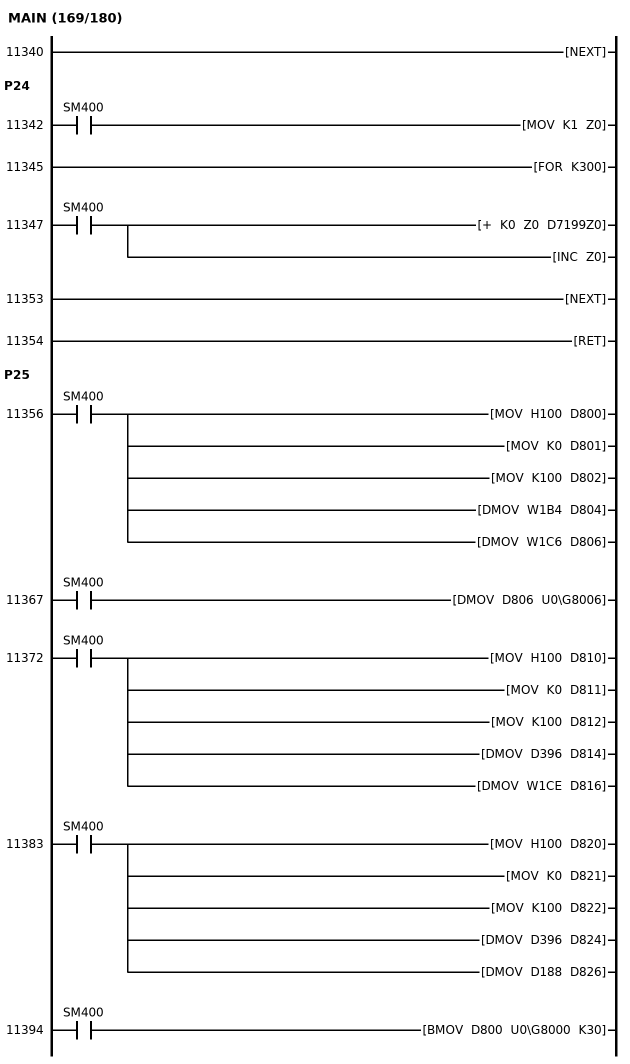
[picture p168: ladder of MAIN, rungs at steps 11340 to 11394]
11340 NEXT
      P24
11342 LD      SM400
      MOV     K1 Z0
11345 FOR     K300
11347 LD      SM400
      +       K0 Z0 D7199Z0
      INC     Z0
11353 NEXT
11354 RET
      P25
11356 LD      SM400
      MOV     H100 D800
      MOV     K0 D801
      MOV     K100 D802
      DMOV    W1B4 D804
      DMOV    W1C6 D806
11367 LD      SM400
      DMOV    D806 U0\G8006
11372 LD      SM400
      MOV     H100 D810
      MOV     K0 D811
      MOV     K100 D812
      DMOV    D396 D814
      DMOV    W1CE D816
11383 LD      SM400
      MOV     H100 D820
      MOV     K0 D821
      MOV     K100 D822
      DMOV    D396 D824
      DMOV    D188 D826
11394 LD      SM400
      BMOV    D800 U0\G8000 K30
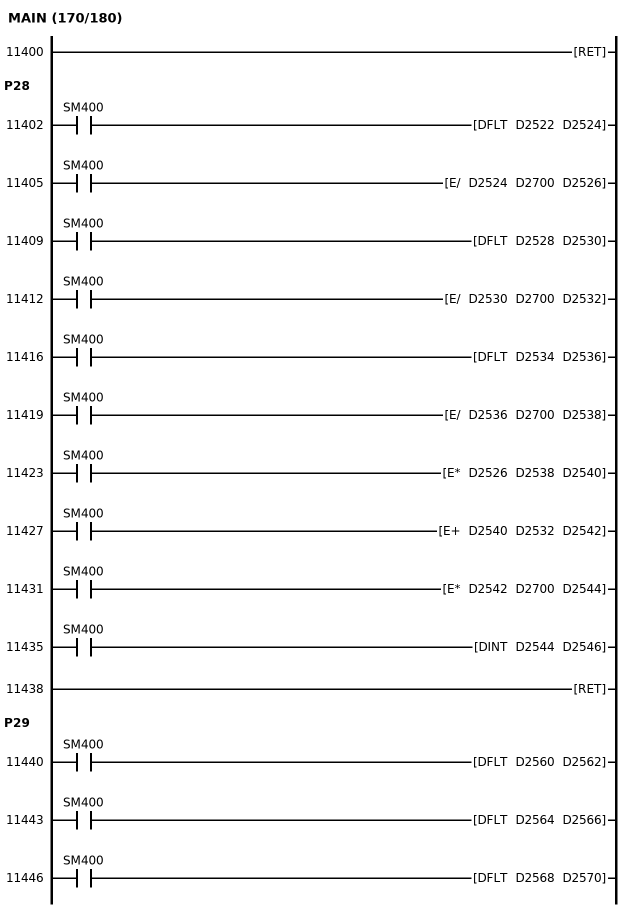
11400 RET
      P28
11402 LD      SM400
      DFLT    D2522 D2524
11405 LD      SM400
      E/      D2524 D2700 D2526
11409 LD      SM400
      DFLT    D2528 D2530
11412 LD      SM400
      E/      D2530 D2700 D2532
11416 LD      SM400
      DFLT    D2534 D2536
11419 LD      SM400
      E/      D2536 D2700 D2538
11423 LD      SM400
      E*      D2526 D2538 D2540
11427 LD      SM400
      E+      D2540 D2532 D2542
11431 LD      SM400
      E*      D2542 D2700 D2544
11435 LD      SM400
      DINT    D2544 D2546
11438 RET
      P29
11440 LD      SM400
      DFLT    D2560 D2562
11443 LD      SM400
      DFLT    D2564 D2566
11446 LD      SM400
      DFLT    D2568 D2570
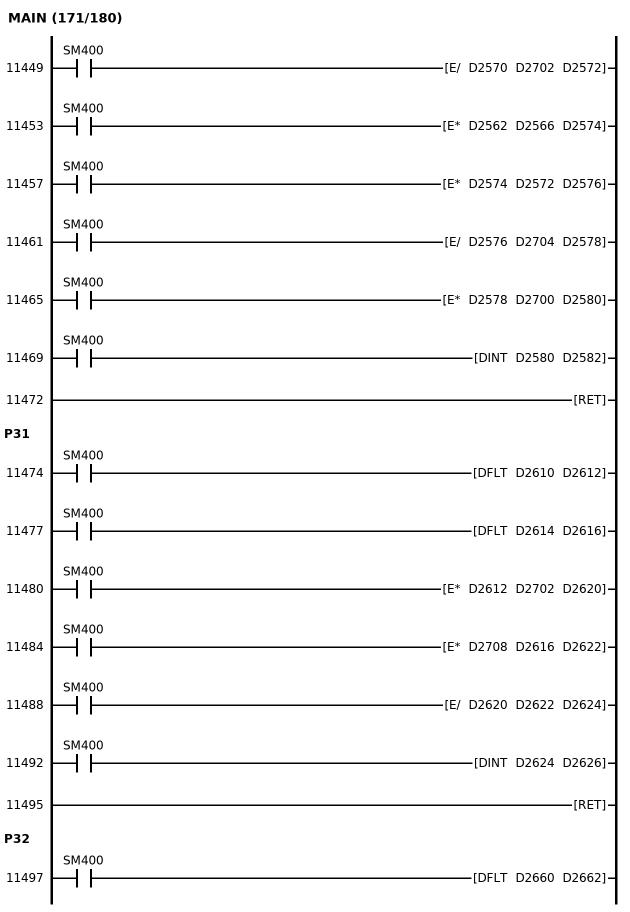
11449 LD      SM400
      E/      D2570 D2702 D2572
11453 LD      SM400
      E*      D2562 D2566 D2574
11457 LD      SM400
      E*      D2574 D2572 D2576
11461 LD      SM400
      E/      D2576 D2704 D2578
11465 LD      SM400
      E*      D2578 D2700 D2580
11469 LD      SM400
      DINT    D2580 D2582
11472 RET
      P31
11474 LD      SM400
      DFLT    D2610 D2612
11477 LD      SM400
      DFLT    D2614 D2616
11480 LD      SM400
      E*      D2612 D2702 D2620
11484 LD      SM400
      E*      D2708 D2616 D2622
11488 LD      SM400
      E/      D2620 D2622 D2624
11492 LD      SM400
      DINT    D2624 D2626
11495 RET
      P32
11497 LD      SM400
      DFLT    D2660 D2662
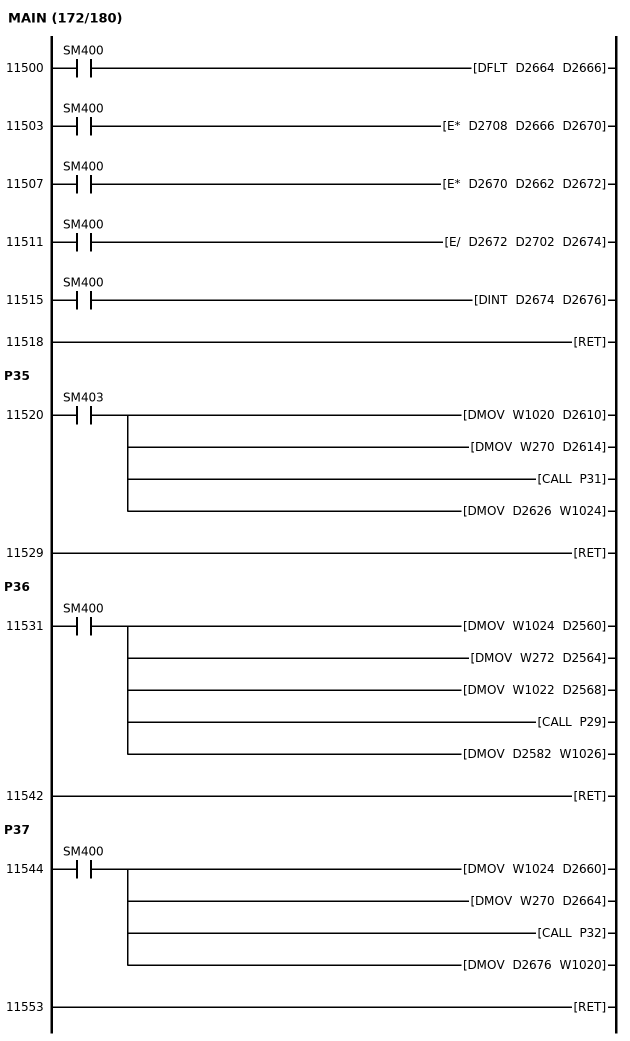
11500 LD      SM400
      DFLT    D2664 D2666
11503 LD      SM400
      E*      D2708 D2666 D2670
11507 LD      SM400
      E*      D2670 D2662 D2672
11511 LD      SM400
      E/      D2672 D2702 D2674
11515 LD      SM400
      DINT    D2674 D2676
11518 RET
      P35
11520 LD      SM403
      DMOV    W1020 D2610
      DMOV    W270 D2614
      CALL    P31
      DMOV    D2626 W1024
11529 RET
      P36
11531 LD      SM400
      DMOV    W1024 D2560
      DMOV    W272 D2564
      DMOV    W1022 D2568
      CALL    P29
      DMOV    D2582 W1026
11542 RET
      P37
11544 LD      SM400
      DMOV    W1024 D2660
      DMOV    W270 D2664
      CALL    P32
      DMOV    D2676 W1020
11553 RET
      P40
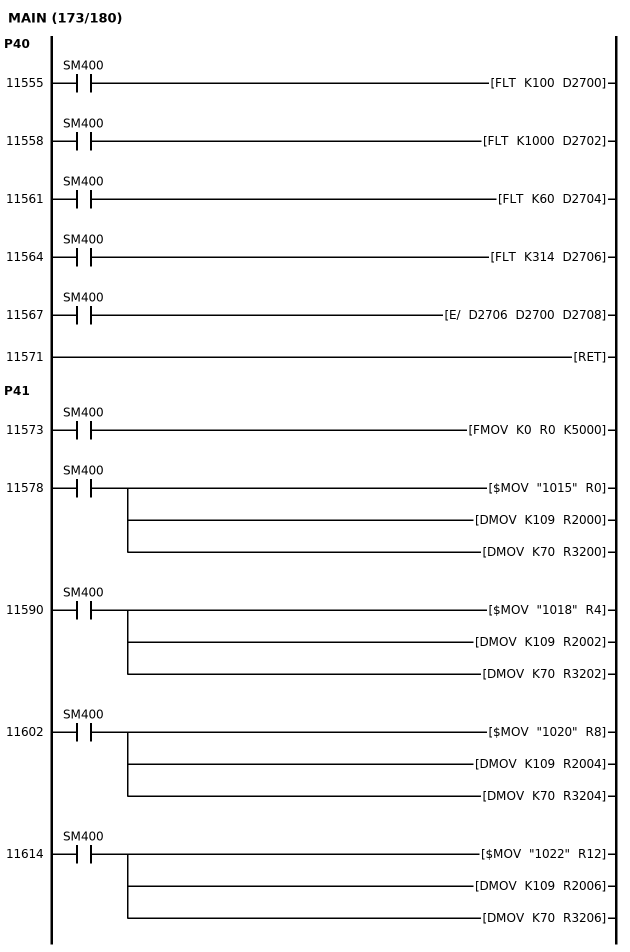
11555 LD      SM400
      FLT     K100 D2700
11558 LD      SM400
      FLT     K1000 D2702
11561 LD      SM400
      FLT     K60 D2704
11564 LD      SM400
      FLT     K314 D2706
11567 LD      SM400
      E/      D2706 D2700 D2708
11571 RET
      P41
11573 LD      SM400
      FMOV    K0 R0 K5000
11578 LD      SM400
      $MOV    "1015" R0
      DMOV    K109 R2000
      DMOV    K70 R3200
11590 LD      SM400
      $MOV    "1018" R4
      DMOV    K109 R2002
      DMOV    K70 R3202
11602 LD      SM400
      $MOV    "1020" R8
      DMOV    K109 R2004
      DMOV    K70 R3204
11614 LD      SM400
      $MOV    "1022" R12
      DMOV    K109 R2006
      DMOV    K70 R3206
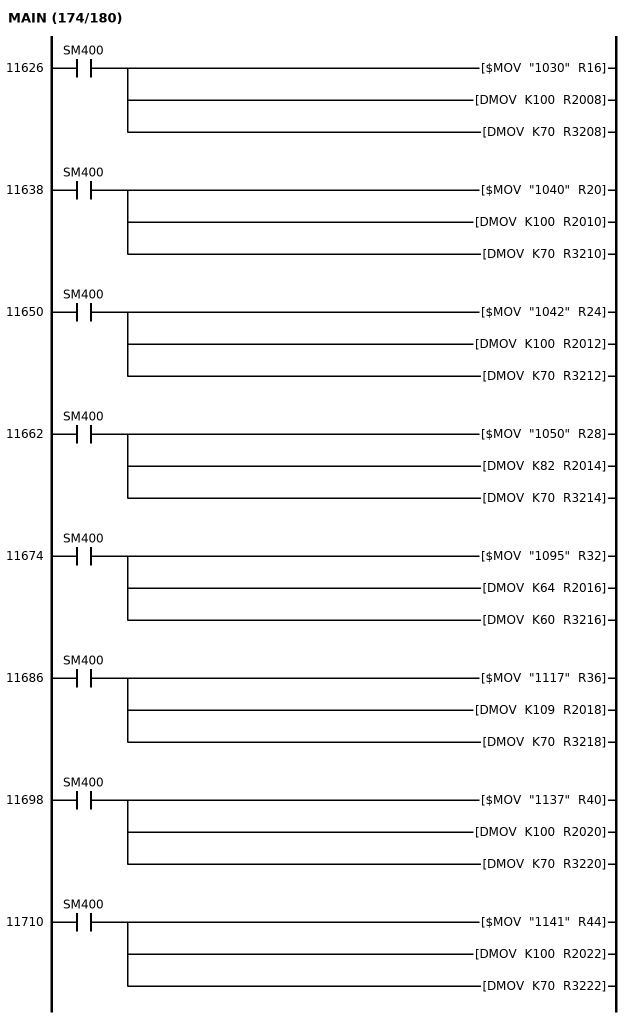
11626 LD      SM400
      $MOV    "1030" R16
      DMOV    K100 R2008
      DMOV    K70 R3208
11638 LD      SM400
      $MOV    "1040" R20
      DMOV    K100 R2010
      DMOV    K70 R3210
11650 LD      SM400
      $MOV    "1042" R24
      DMOV    K100 R2012
      DMOV    K70 R3212
11662 LD      SM400
      $MOV    "1050" R28
      DMOV    K82 R2014
      DMOV    K70 R3214
11674 LD      SM400
      $MOV    "1095" R32
      DMOV    K64 R2016
      DMOV    K60 R3216
11686 LD      SM400
      $MOV    "1117" R36
      DMOV    K109 R2018
      DMOV    K70 R3218
11698 LD      SM400
      $MOV    "1137" R40
      DMOV    K100 R2020
      DMOV    K70 R3220
11710 LD      SM400
      $MOV    "1141" R44
      DMOV    K100 R2022
      DMOV    K70 R3222
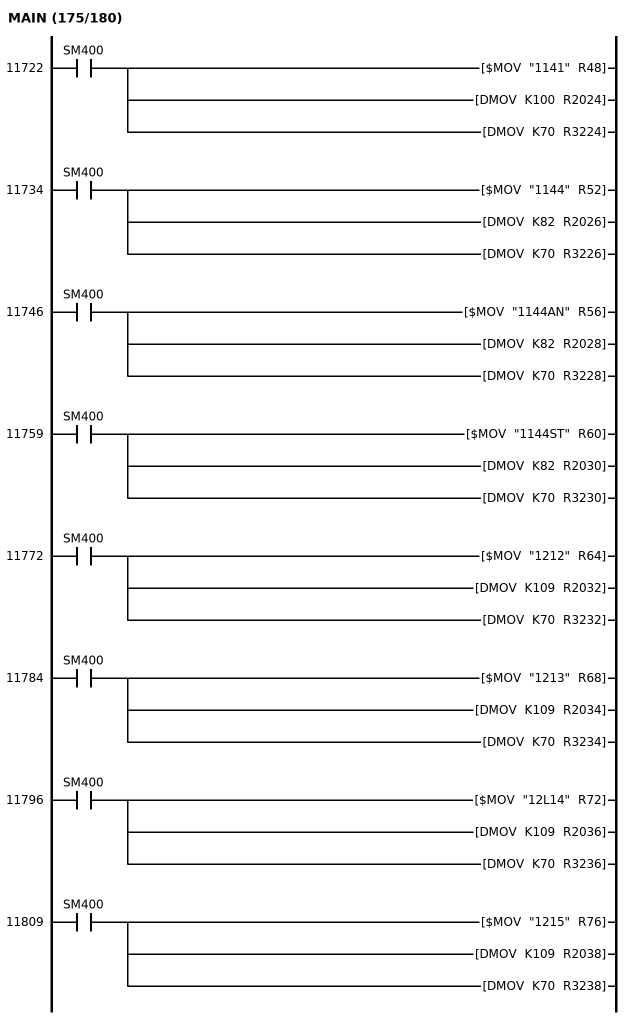
11722 LD      SM400
      $MOV    "1141" R48
      DMOV    K100 R2024
      DMOV    K70 R3224
11734 LD      SM400
      $MOV    "1144" R52
      DMOV    K82 R2026
      DMOV    K70 R3226
11746 LD      SM400
      $MOV    "1144AN" R56
      DMOV    K82 R2028
      DMOV    K70 R3228
11759 LD      SM400
      $MOV    "1144ST" R60
      DMOV    K82 R2030
      DMOV    K70 R3230
11772 LD      SM400
      $MOV    "1212" R64
      DMOV    K109 R2032
      DMOV    K70 R3232
11784 LD      SM400
      $MOV    "1213" R68
      DMOV    K109 R2034
      DMOV    K70 R3234
11796 LD      SM400
      $MOV    "12L14" R72
      DMOV    K109 R2036
      DMOV    K70 R3236
11809 LD      SM400
      $MOV    "1215" R76
      DMOV    K109 R2038
      DMOV    K70 R3238
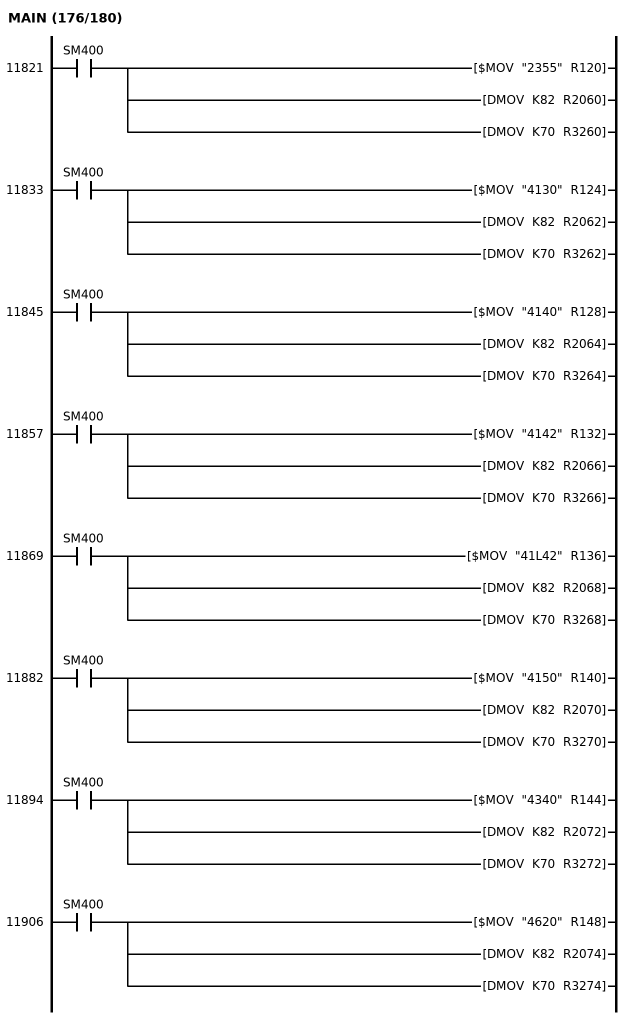
11821 LD      SM400
      $MOV    "2355" R120
      DMOV    K82 R2060
      DMOV    K70 R3260
11833 LD      SM400
      $MOV    "4130" R124
      DMOV    K82 R2062
      DMOV    K70 R3262
11845 LD      SM400
      $MOV    "4140" R128
      DMOV    K82 R2064
      DMOV    K70 R3264
11857 LD      SM400
      $MOV    "4142" R132
      DMOV    K82 R2066
      DMOV    K70 R3266
11869 LD      SM400
      $MOV    "41L42" R136
      DMOV    K82 R2068
      DMOV    K70 R3268
11882 LD      SM400
      $MOV    "4150" R140
      DMOV    K82 R2070
      DMOV    K70 R3270
11894 LD      SM400
      $MOV    "4340" R144
      DMOV    K82 R2072
      DMOV    K70 R3272
11906 LD      SM400
      $MOV    "4620" R148
      DMOV    K82 R2074
      DMOV    K70 R3274
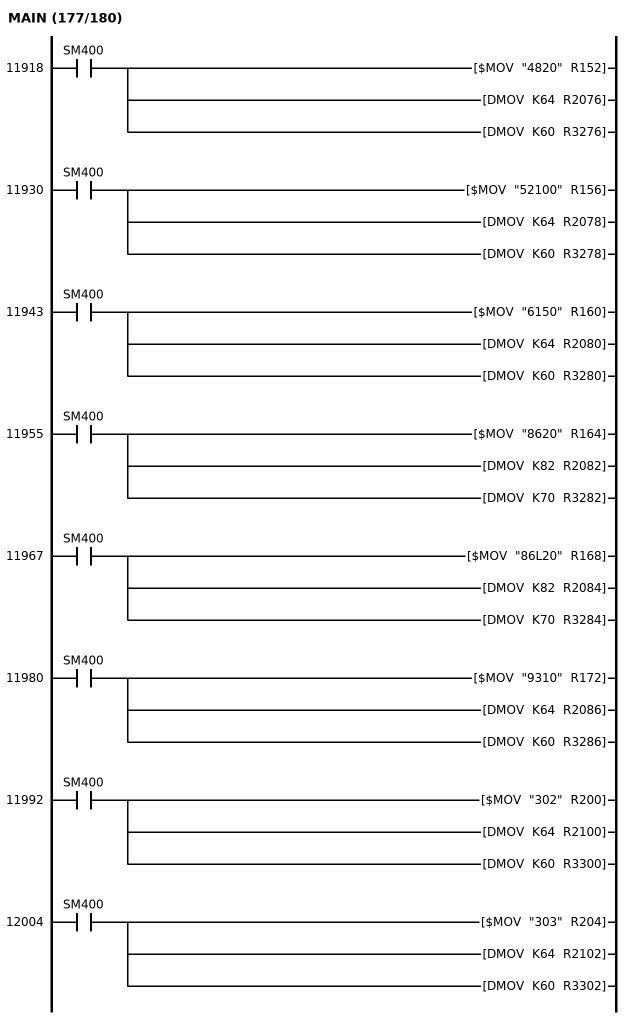
11918 LD      SM400
      $MOV    "4820" R152
      DMOV    K64 R2076
      DMOV    K60 R3276
11930 LD      SM400
      $MOV    "52100" R156
      DMOV    K64 R2078
      DMOV    K60 R3278
11943 LD      SM400
      $MOV    "6150" R160
      DMOV    K64 R2080
      DMOV    K60 R3280
11955 LD      SM400
      $MOV    "8620" R164
      DMOV    K82 R2082
      DMOV    K70 R3282
11967 LD      SM400
      $MOV    "86L20" R168
      DMOV    K82 R2084
      DMOV    K70 R3284
11980 LD      SM400
      $MOV    "9310" R172
      DMOV    K64 R2086
      DMOV    K60 R3286
11992 LD      SM400
      $MOV    "302" R200
      DMOV    K64 R2100
      DMOV    K60 R3300
12004 LD      SM400
      $MOV    "303" R204
      DMOV    K64 R2102
      DMOV    K60 R3302
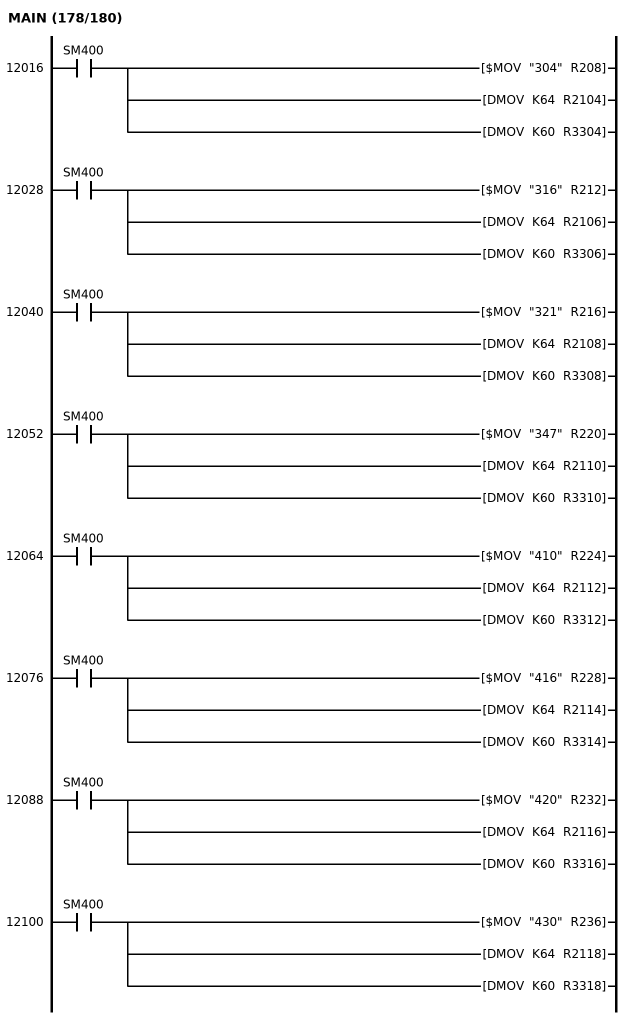
12016 LD      SM400
      $MOV    "304" R208
      DMOV    K64 R2104
      DMOV    K60 R3304
12028 LD      SM400
      $MOV    "316" R212
      DMOV    K64 R2106
      DMOV    K60 R3306
12040 LD      SM400
      $MOV    "321" R216
      DMOV    K64 R2108
      DMOV    K60 R3308
12052 LD      SM400
      $MOV    "347" R220
      DMOV    K64 R2110
      DMOV    K60 R3310
12064 LD      SM400
      $MOV    "410" R224
      DMOV    K64 R2112
      DMOV    K60 R3312
12076 LD      SM400
      $MOV    "416" R228
      DMOV    K64 R2114
      DMOV    K60 R3314
12088 LD      SM400
      $MOV    "420" R232
      DMOV    K64 R2116
      DMOV    K60 R3316
12100 LD      SM400
      $MOV    "430" R236
      DMOV    K64 R2118
      DMOV    K60 R3318
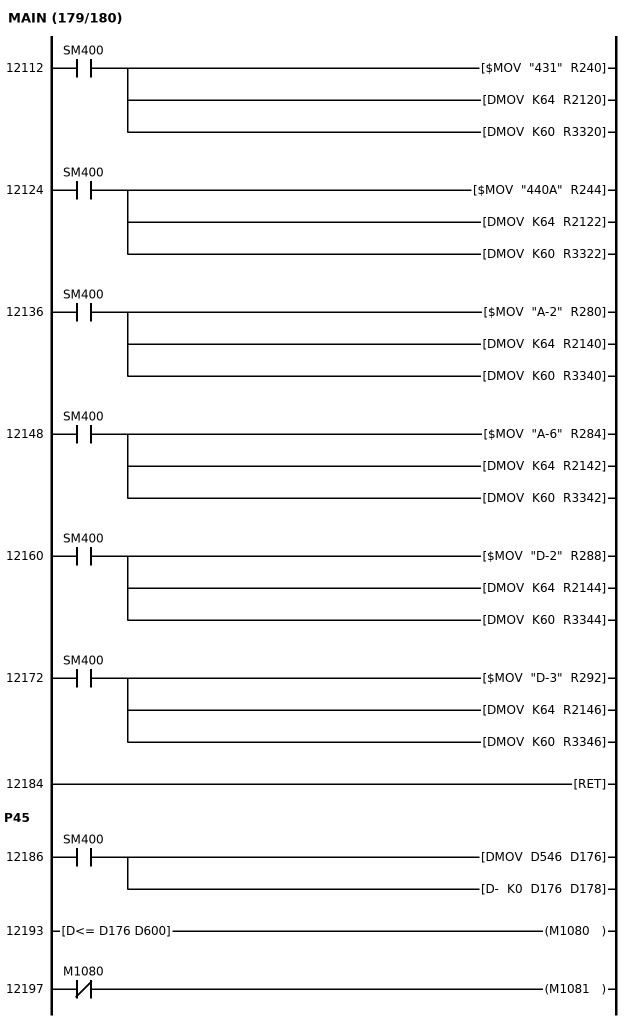
12112 LD      SM400
      $MOV    "431" R240
      DMOV    K64 R2120
      DMOV    K60 R3320
12124 LD      SM400
      $MOV    "440A" R244
      DMOV    K64 R2122
      DMOV    K60 R3322
12136 LD      SM400
      $MOV    "A-2" R280
      DMOV    K64 R2140
      DMOV    K60 R3340
12148 LD      SM400
      $MOV    "A-6" R284
      DMOV    K64 R2142
      DMOV    K60 R3342
12160 LD      SM400
      $MOV    "D-2" R288
      DMOV    K64 R2144
      DMOV    K60 R3344
12172 LD      SM400
      $MOV    "D-3" R292
      DMOV    K64 R2146
      DMOV    K60 R3346
12184 RET
      P45
12186 LD      SM400
      DMOV    D546 D176
      D-      K0 D176 D178
12193 LDD<=   D176 D600
      OUT     M1080
12197 LDI     M1080
      OUT     M1081
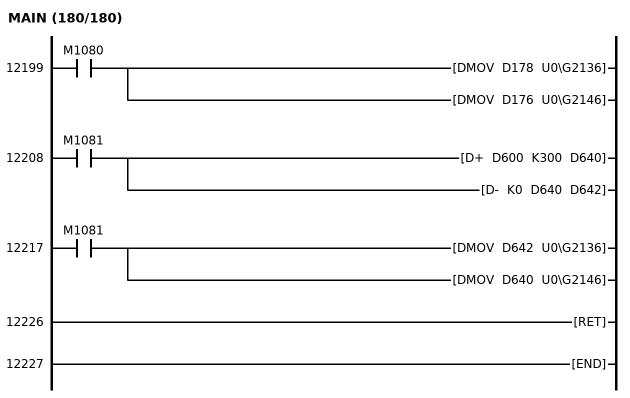
12199 LD      M1080
      DMOV    D178 U0\G2136
      DMOV    D176 U0\G2146
12208 LD      M1081
      D+      D600 K300 D640
      D-      K0 D640 D642
12217 LD      M1081
      DMOV    D642 U0\G2136
      DMOV    D640 U0\G2146
12226 RET
12227 END
END_PROGRAM

PROGRAM HMS
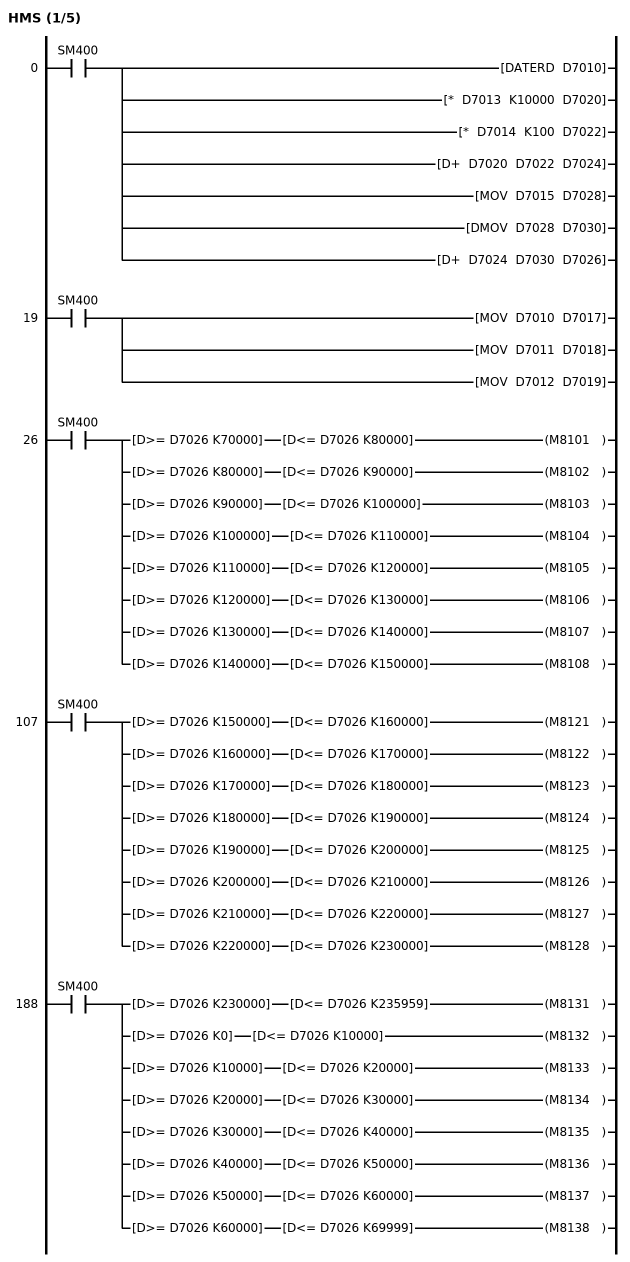
0     LD      SM400
      DATERD  D7010
      *       D7013 K10000 D7020
      *       D7014 K100 D7022
      D+      D7020 D7022 D7024
      MOV     D7015 D7028
      DMOV    D7028 D7030
      D+      D7024 D7030 D7026
19    LD      SM400
      MOV     D7010 D7017
      MOV     D7011 D7018
      MOV     D7012 D7019
26    LD      SM400
      MPS
      ANDD>=  D7026 K70000
      ANDD<=  D7026 K80000
      OUT     M8101
      MRD
      ANDD>=  D7026 K80000
      ANDD<=  D7026 K90000
      OUT     M8102
      MRD
      ANDD>=  D7026 K90000
      ANDD<=  D7026 K100000
      OUT     M8103
      MRD
      ANDD>=  D7026 K100000
      ANDD<=  D7026 K110000
      OUT     M8104
      MRD
      ANDD>=  D7026 K110000
      ANDD<=  D7026 K120000
      OUT     M8105
      MRD
      ANDD>=  D7026 K120000
      ANDD<=  D7026 K130000
      OUT     M8106
      MRD
      ANDD>=  D7026 K130000
      ANDD<=  D7026 K140000
      OUT     M8107
      MPP
      ANDD>=  D7026 K140000
      ANDD<=  D7026 K150000
      OUT     M8108
107   LD      SM400
      MPS
      ANDD>=  D7026 K150000
      ANDD<=  D7026 K160000
      OUT     M8121
      MRD
      ANDD>=  D7026 K160000
      ANDD<=  D7026 K170000
      OUT     M8122
      MRD
      ANDD>=  D7026 K170000
      ANDD<=  D7026 K180000
      OUT     M8123
      MRD
      ANDD>=  D7026 K180000
      ANDD<=  D7026 K190000
      OUT     M8124
      MRD
      ANDD>=  D7026 K190000
      ANDD<=  D7026 K200000
      OUT     M8125
      MRD
      ANDD>=  D7026 K200000
      ANDD<=  D7026 K210000
      OUT     M8126
      MRD
      ANDD>=  D7026 K210000
      ANDD<=  D7026 K220000
      OUT     M8127
      MPP
      ANDD>=  D7026 K220000
      ANDD<=  D7026 K230000
      OUT     M8128
188   LD      SM400
      MPS
      ANDD>=  D7026 K230000
      ANDD<=  D7026 K235959
      OUT     M8131
      MRD
      ANDD>=  D7026 K0
      ANDD<=  D7026 K10000
      OUT     M8132
      MRD
      ANDD>=  D7026 K10000
      ANDD<=  D7026 K20000
      OUT     M8133
      MRD
      ANDD>=  D7026 K20000
      ANDD<=  D7026 K30000
      OUT     M8134
      MRD
      ANDD>=  D7026 K30000
      ANDD<=  D7026 K40000
      OUT     M8135
      MRD
      ANDD>=  D7026 K40000
      ANDD<=  D7026 K50000
      OUT     M8136
      MRD
      ANDD>=  D7026 K50000
      ANDD<=  D7026 K60000
      OUT     M8137
      MPP
      ANDD>=  D7026 K60000
      ANDD<=  D7026 K69999
      OUT     M8138
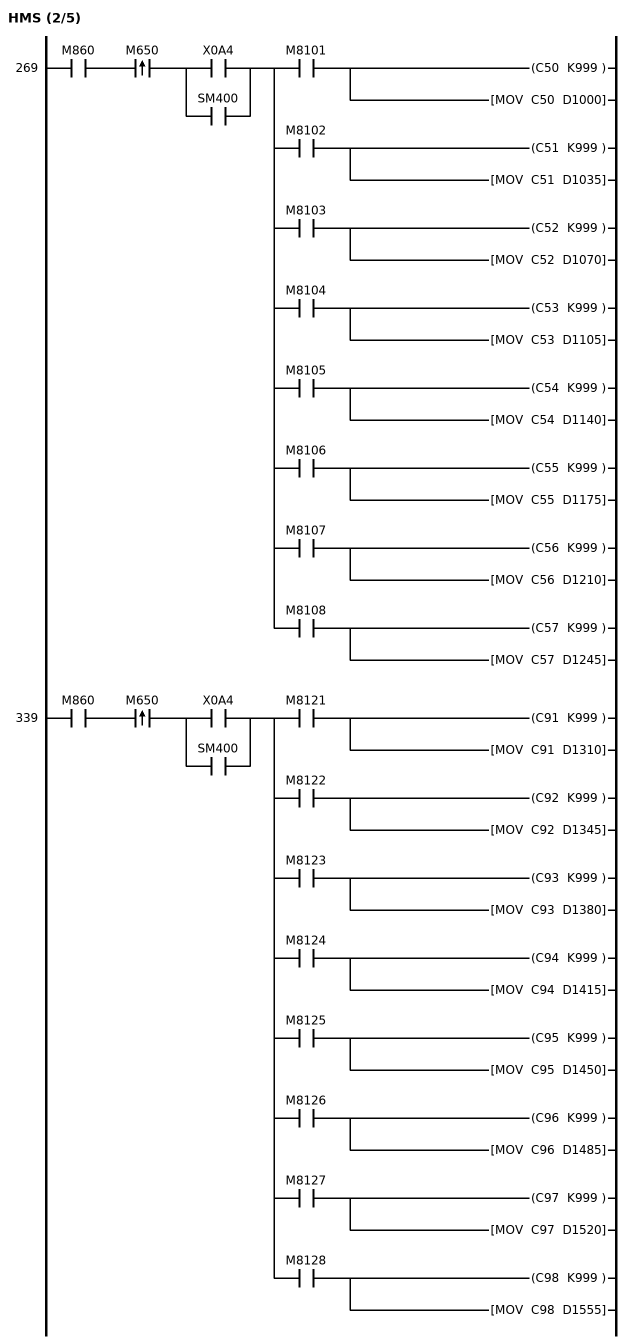
269   LD      M860
      ANDP    M650
      LD      X0A4
      OR      SM400
      ANB
      MPS
      AND     M8101
      OUT     C50 K999
      MOV     C50 D1000
      MRD
      AND     M8102
      OUT     C51 K999
      MOV     C51 D1035
      MRD
      AND     M8103
      OUT     C52 K999
      MOV     C52 D1070
      MRD
      AND     M8104
      OUT     C53 K999
      MOV     C53 D1105
      MRD
      AND     M8105
      OUT     C54 K999
      MOV     C54 D1140
      MRD
      AND     M8106
      OUT     C55 K999
      MOV     C55 D1175
      MRD
      AND     M8107
      OUT     C56 K999
      MOV     C56 D1210
      MPP
      AND     M8108
      OUT     C57 K999
      MOV     C57 D1245
339   LD      M860
      ANDP    M650
      LD      X0A4
      OR      SM400
      ANB
      MPS
      AND     M8121
      OUT     C91 K999
      MOV     C91 D1310
      MRD
      AND     M8122
      OUT     C92 K999
      MOV     C92 D1345
      MRD
      AND     M8123
      OUT     C93 K999
      MOV     C93 D1380
      MRD
      AND     M8124
      OUT     C94 K999
      MOV     C94 D1415
      MRD
      AND     M8125
      OUT     C95 K999
      MOV     C95 D1450
      MRD
      AND     M8126
      OUT     C96 K999
      MOV     C96 D1485
      MRD
      AND     M8127
      OUT     C97 K999
      MOV     C97 D1520
      MPP
      AND     M8128
      OUT     C98 K999
      MOV     C98 D1555
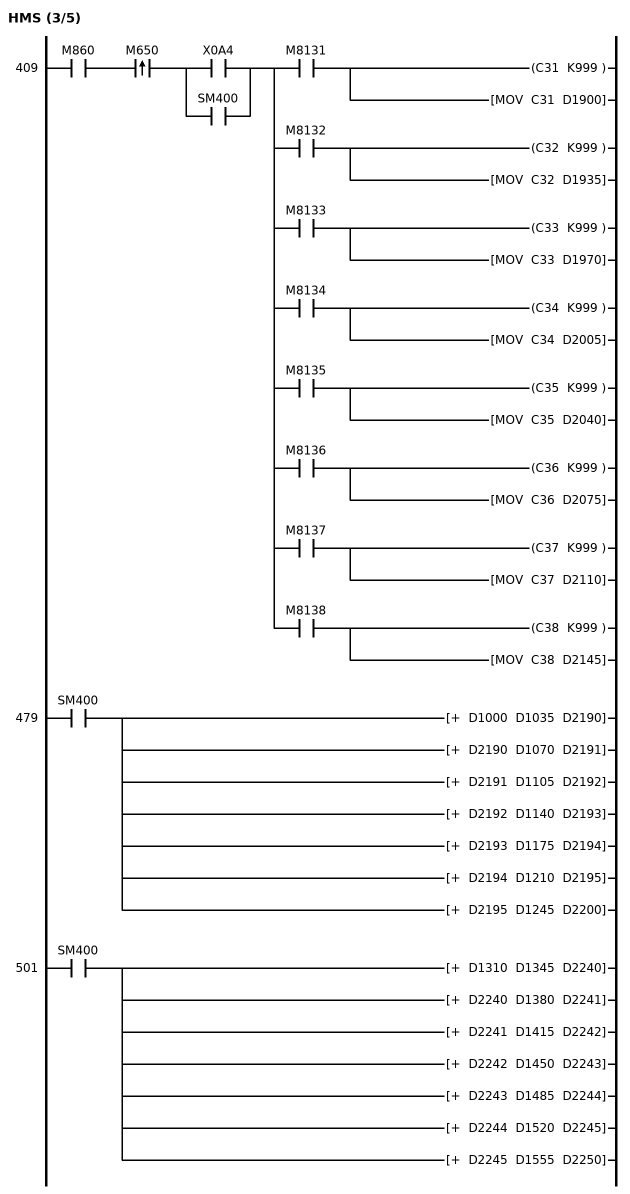
409   LD      M860
      ANDP    M650
      LD      X0A4
      OR      SM400
      ANB
      MPS
      AND     M8131
      OUT     C31 K999
      MOV     C31 D1900
      MRD
      AND     M8132
      OUT     C32 K999
      MOV     C32 D1935
      MRD
      AND     M8133
      OUT     C33 K999
      MOV     C33 D1970
      MRD
      AND     M8134
      OUT     C34 K999
      MOV     C34 D2005
      MRD
      AND     M8135
      OUT     C35 K999
      MOV     C35 D2040
      MRD
      AND     M8136
      OUT     C36 K999
      MOV     C36 D2075
      MRD
      AND     M8137
      OUT     C37 K999
      MOV     C37 D2110
      MPP
      AND     M8138
      OUT     C38 K999
      MOV     C38 D2145
479   LD      SM400
      +       D1000 D1035 D2190
      +       D2190 D1070 D2191
      +       D2191 D1105 D2192
      +       D2192 D1140 D2193
      +       D2193 D1175 D2194
      +       D2194 D1210 D2195
      +       D2195 D1245 D2200
501   LD      SM400
      +       D1310 D1345 D2240
      +       D2240 D1380 D2241
      +       D2241 D1415 D2242
      +       D2242 D1450 D2243
      +       D2243 D1485 D2244
      +       D2244 D1520 D2245
      +       D2245 D1555 D2250
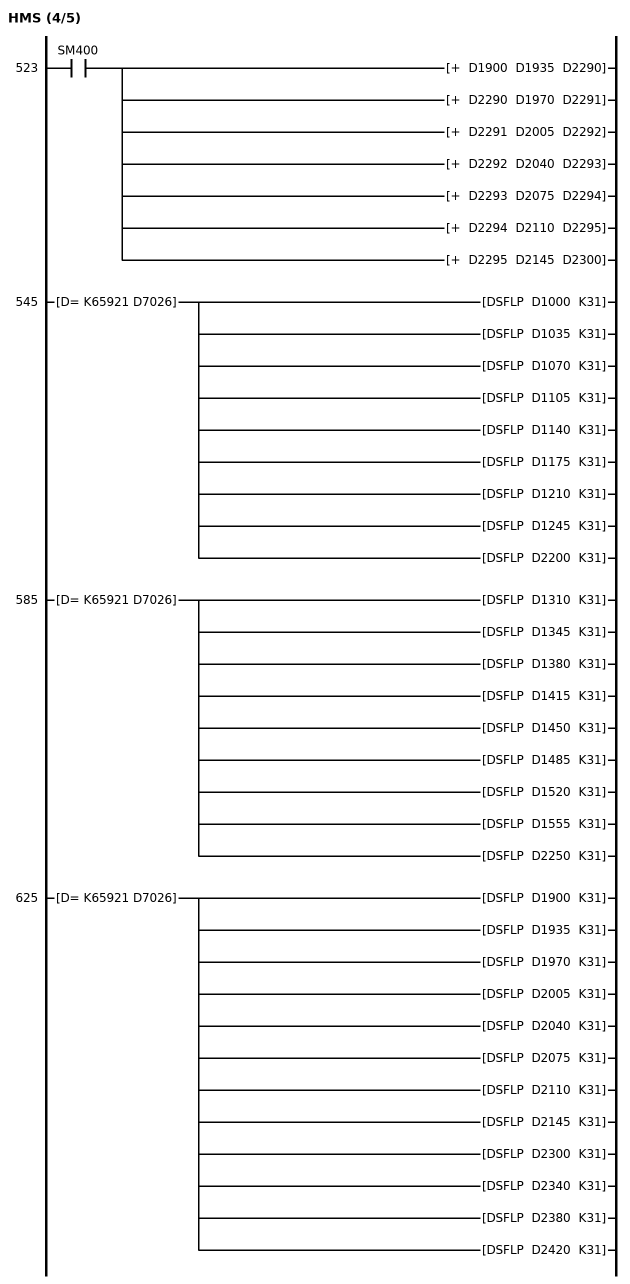
523   LD      SM400
      +       D1900 D1935 D2290
      +       D2290 D1970 D2291
      +       D2291 D2005 D2292
      +       D2292 D2040 D2293
      +       D2293 D2075 D2294
      +       D2294 D2110 D2295
      +       D2295 D2145 D2300
545   LDD=    K65921 D7026
      DSFLP   D1000 K31
      DSFLP   D1035 K31
      DSFLP   D1070 K31
      DSFLP   D1105 K31
      DSFLP   D1140 K31
      DSFLP   D1175 K31
      DSFLP   D1210 K31
      DSFLP   D1245 K31
      DSFLP   D2200 K31
585   LDD=    K65921 D7026
      DSFLP   D1310 K31
      DSFLP   D1345 K31
      DSFLP   D1380 K31
      DSFLP   D1415 K31
      DSFLP   D1450 K31
      DSFLP   D1485 K31
      DSFLP   D1520 K31
      DSFLP   D1555 K31
      DSFLP   D2250 K31
625   LDD=    K65921 D7026
      DSFLP   D1900 K31
      DSFLP   D1935 K31
      DSFLP   D1970 K31
      DSFLP   D2005 K31
      DSFLP   D2040 K31
      DSFLP   D2075 K31
      DSFLP   D2110 K31
      DSFLP   D2145 K31
      DSFLP   D2300 K31
      DSFLP   D2340 K31
      DSFLP   D2380 K31
      DSFLP   D2420 K31
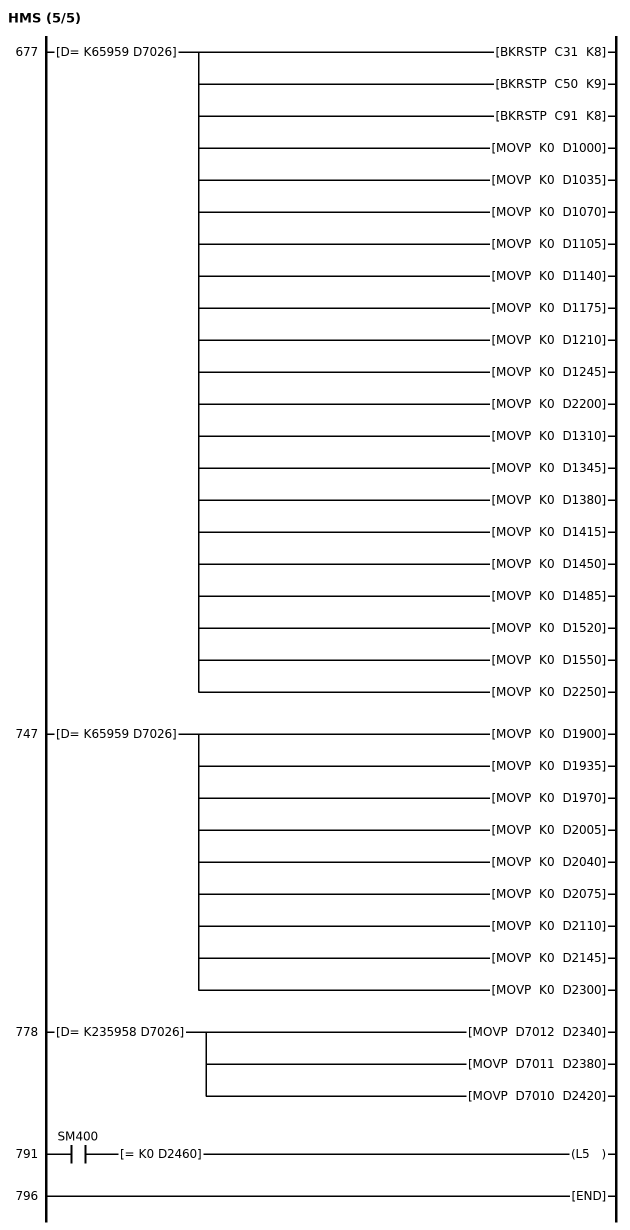
677   LDD=    K65959 D7026
      BKRSTP  C31 K8
      BKRSTP  C50 K9
      BKRSTP  C91 K8
      MOVP    K0 D1000
      MOVP    K0 D1035
      MOVP    K0 D1070
      MOVP    K0 D1105
      MOVP    K0 D1140
      MOVP    K0 D1175
      MOVP    K0 D1210
      MOVP    K0 D1245
      MOVP    K0 D2200
      MOVP    K0 D1310
      MOVP    K0 D1345
      MOVP    K0 D1380
      MOVP    K0 D1415
      MOVP    K0 D1450
      MOVP    K0 D1485
      MOVP    K0 D1520
      MOVP    K0 D1550
      MOVP    K0 D2250
747   LDD=    K65959 D7026
      MOVP    K0 D1900
      MOVP    K0 D1935
      MOVP    K0 D1970
      MOVP    K0 D2005
      MOVP    K0 D2040
      MOVP    K0 D2075
      MOVP    K0 D2110
      MOVP    K0 D2145
      MOVP    K0 D2300
778   LDD=    K235958 D7026
      MOVP    D7012 D2340
      MOVP    D7011 D2380
      MOVP    D7010 D2420
791   LD      SM400
      AND=    K0 D2460
      OUT     L5
796   END
END_PROGRAM
